FUNCTION_BLOCK FB_Delay
VAR_INPUT
	msec:INT;
END_VAR
VAR_OUTPUT
END_VAR
VAR
	tim:TON;
END_VAR
VAR_IN_OUT
	in:BOOL;
	out:BOOL;
END_VAR

tim(IN:=in,PT:=INT_TO_TIME(msec));
out:=tim.Q;

END_FUNCTION_BLOCK

(* stored: Version 1.1.0.1, ProductVersion 3.1.4022.18
   POU FB_Delay: Id {ae206355-42b6-443f-8e61-84262bc80476}, SpecialFunc None *)
